// TIA Portal V17 export
// export: Created 2024-09-02T12:50:17.7134452Z, ExportSetting WithDefaults, DisplayName Totally Integrated Automation Portal, DisplayVersion V17, DisplayName TIA Portal Openness, DisplayVersion V17, DisplayName TIA Portal Version Control Interface, DisplayVersion V17, DisplayName STEP 7 Professional, DisplayVersion V17, DisplayName STEP 7 Safety, DisplayVersion V17, DisplayName WinCC Professional, DisplayVersion V17
DATA_BLOCK "SysDB_ZP_SeriesError_OP70"   // DB268
{ S7_Optimized_Access := 'TRUE'; DB_Accessible_From_OPC_UA := 'FALSE' }
AUTHOR : OlegFuehrus
FAMILY : BA
NAME : BA
VERSION : 0.1
// stored: AutoNumber true, DBAccessibleFromOPCUA false, IsOnlyStoredInLoadMemory false, IsRetainMemResEnabled false, IsWriteProtectedInAS false, MemoryReserve 100
   VAR RETAIN
      SeriesError { S7_SetPoint := 'True'} : Array[1..64] of "TypeSeriesError";
   END_VAR
BEGIN
END_DATA_BLOCK
